PROGRAM MAIN
VAR
	OpenFlap:	BOOL;
	CloseFlap:	BOOL;
	OpenSlit:	BOOL;
	CloseSlit:	BOOL;
	FlapOpen:	BOOL := FALSE;
	FlapClosed:	BOOL := FALSE;
	SlitOpen:	BOOL := FALSE;
	SlitClosed:	BOOL := FALSE;
	// assume dome open, after power loss / reboot
	DomeOpen:	BOOL := TRUE;
	DomeClosed:	BOOL := FALSE;
	FlapDelay,
	SlitDelay:	TON;
	FlapTimer,
	SlitTimer:	TP;
	FlapDone,
	SlitDone:	F_TRIG;
	SyncOut:	TON;
	TimeOut:	TON;
	WD_LED:		E_CX81x0_LED;
	ERR_LED:	E_CX81x0_LED;
	(*
	Serial: MDP5001_600_C98F2494;
	SerialLineControl: SerialLineControl;
	SerialError: INT;
	RxBuffer,
	TxBuffer: ComBuffer;
	*)
END_VAR

(*
Dome Control Remote Unit CX8190
########################

The dome is controlled by the main PLC using the GVL_Dome.ControlWord,
which is used to exchange commands to open and close the slit and the flap
and to report wether the dome is open or closed.
*)
IF GVL_Dome.ControlWord.0 THEN // we have valid data
	OpenFlap := GVL_Dome.ControlWord.1;
	OpenSlit := GVL_Dome.ControlWord.2;
	CloseFlap := NOT GVL_Dome.ControlWord.1;
	CloseSlit := NOT GVL_Dome.ControlWord.2;
	ERR_LED := E_CX81x0_LED.eCX81x0_LED_RED_OFF;
END_IF

// This is the sync timeout. If we loose the sync for 5 seconds, we issue a warning.
SyncOut(IN := NOT GVL_Dome.ControlWord.0, PT := T#5S);
IF SyncOut.Q THEN
	ERR_LED := E_CX81x0_LED.eCX81x0_LED_RED_FLASHING_200ms;
END_IF

// This is the watchdog timer. If we don't get a valid signal within n seconds, we issue to close the dome.
TimeOut(IN := NOT GVL_Dome.ControlWord.0, PT := T#30S);
IF TimeOut.Q THEN
	CloseFlap := TRUE;
	CloseSlit := TRUE;
	ERR_LED := E_CX81x0_LED.eCX81x0_LED_RED_ON;
END_IF

// cancel commands, if we know that the slot is closed
IF SlitClosed AND CloseSlit THEN
	CloseSlit := FALSE;
END_IF
IF SlitOpen AND OpenSlit THEN
	OpenSlit := FALSE;
END_IF
IF FlapClosed AND CloseFlap THEN
	CloseFlap := FALSE;
END_IF
IF FlapOpen AND OpenFlap THEN
	OpenFlap := FALSE;
END_IF

IF CloseSlit THEN
	OpenSlit := FALSE;
	GVL_Dome.Slit_open := FALSE;
	WD_LED := E_CX81x0_LED.eCX81x0_LED_GREEN_FLASHING_500ms;
END_IF

IF OpenSlit THEN
	GVL_Dome.Slit_open := TRUE;
	WD_LED := E_CX81x0_LED.eCX81x0_LED_RED_FLASHING_500ms;
END_IF

IF CloseFlap THEN
	OpenFlap := FALSE;
	GVL_Dome.Flap_open := FALSE;
	WD_LED := E_CX81x0_LED.eCX81x0_LED_GREEN_FLASHING_200ms;
END_IF

IF OpenFlap THEN
	GVL_Dome.Flap_open := TRUE;
	WD_LED := E_CX81x0_LED.eCX81x0_LED_RED_FLASHING_200ms;
END_IF

// if we reverse the direction of the flap, wait n milliseconds, otherwise we blow the fuse
FlapDelay(  IN := OpenFlap OR CloseFlap,
			PT := T#1000MS);
// After an initial delay, enable the signal for n seconds to move the flap.			
FlapTimer(  IN := FlapDelay.Q,
			PT := T#30S,
			Q => GVL_Dome.Flap_enable);
// a falling edge of the enable signal indicates, that we are done
FlapDone(CLK := GVL_Dome.Flap_enable);
// deactivate open or close signal if enable becomes false;
IF FlapDone.Q THEN
	IF OpenFlap THEN
		FlapOpen 	:= TRUE;
		FlapClosed 	:= FALSE;
	ELSIF CloseFlap THEN
		FlapClosed 	:= TRUE;
		FlapOpen 	:= FALSE;
	END_IF
	OpenFlap := FALSE;
	CloseFlap := FALSE;
END_IF
			
// if we reverse the direction of the flap, wait n milliseconds, otherwise we blow the fuse
SlitDelay(  IN := OpenSlit OR CloseSlit, 
			PT := T#1000MS); 

// After an initial delay, enable the signal for n seconds to move the slit.			
SlitTimer(  IN := SlitDelay.Q,
			PT := T#70S,
			Q => GVL_Dome.Slit_enable); 
// a falling edge of the enable signal indicates, that we are done			
SlitDone(CLK := GVL_Dome.Slit_enable);

IF SlitDone.Q THEN
	IF OpenSlit THEN
		SlitOpen := TRUE;
	ELSIF CloseSlit THEN
		SlitClosed := TRUE;
	END_IF
	OpenSlit := FALSE;
	CloseSlit := FALSE;
END_IF

IF DomeOpen THEN
	WD_LED := E_CX81x0_LED.eCX81x0_LED_RED_ON;
END_IF
IF DomeClosed THEN
	WD_LED := E_CX81x0_LED.eCX81x0_LED_GREEN_ON;
END_IF

DomeOpen := FlapOpen AND SlitOpen;
DomeClosed := FlapClosed AND SlitClosed;

F_CX8190_LED_WD(eMode := WD_LED);
F_CX8190_LED_ERR(eMode := ERR_LED);

// reset the controlword
GVL_Dome.ControlWord.0 := 0;
GVL_Dome.ControlWord.3 := DomeOpen;
GVL_Dome.ControlWord.4 := DomeClosed;

(*
SerialLineControl(Mode := ComSerialLineMode_t.SERIALLINEMODE_EL6_22B,
	pComIn := ADR(Serial.MDP5001_600_Input.MDP5001_600_COM_TxPDO_Map_Inputs_Data_In_0),
	pComOut := ADR(Serial.MDP5001_600_Output.MDP5001_600_COM_RxPDO_Map_Outputs_Data_Out_0),
	ErrorID => SerialError,
	TxBuffer := Txbuffer,
	RxBuffer := RxBuffer
	);
*)

END_PROGRAM

(* stored: Version 1.1.0.1, ProductVersion 3.1.4024.6
   POU MAIN: Id {7c90e337-da70-41ec-ab5c-8c28e27e5b13}, SpecialFunc None *)
